// TIA Portal project "Su Tankının Doldurulup Boşaltılması_V15.1" (V15.1)
// Vorlageprojekt für das Buch mit Zielsystem S7-1200

(* hardware
DEVICE "S7-1200-Station_1"  S7-1200 Station
   slot 0: "Baugruppenträger_0"  Rack  V1.0
   slot 1: "PLC_1"  CPU 1212C DC/DC/DC  6ES7 212-1AE40-0XB0  V4.2
   slot 2: "AI 4x13BIT/AQ 2x14BIT_1"  6ES7 234-4HE32-0XB0  V2.0
DEVICE "PC-System_1"  SIMATIC PC station
   slot 0: "SIMATIC PC station"  Rail  SIMATIC PC-Station  V1.0
      slot 125: "Stationmanager"  Station_Manager  V6.0.4
   slot 1: "HMI_RT_1"  WinCC RT Advanced  6AV2 104-0xxxx-xxxx  15.1.0.0
      slot 33792: "Host interface"  Host interface
   slot 2: "IE general_1"  IE General  IE_CP  V8.2.0
*)

// ===== PLC "PLC_1"  CPU 1212C DC/DC/DC =====

VAR_GLOBAL   // PLC tag table "PLC_TAGS"
   "stop_button" AT %I0.0 : Bool;
   "start_button" AT %I0.1 : Bool;
   "sistem_devrede" AT %M5.0 : Bool;
   "set_reset_mem" AT %M5.1 : Bool;
   "sıvı_seviyesi_sensor" AT %IW30 : Int;
   "sıvı_basıncı_sensor" AT %IW32 : Int;
   "sıvı_ekle_butonu" AT %I0.3 : Bool;
   "sıvı_bosalt_butonu" AT %I0.4 : Bool;
   "Tag_1" AT %M7.1 : Bool;
   "Tag_2" AT %M7.5 : Bool;
   "Tag_3" AT %M9.0 : Bool;
END_VAR

VAR_GLOBAL   // PLC tag table "HMI_TAGS"
   "HMI_stop" AT %M6.0 : Bool;
   "HMI_start" AT %M6.1 : Bool;
   "hmi_vana_ekle" AT %QW30 : Int;
   "hmi_boşalt_boşalt" AT %QW32 : Int;
   "hmi_sıvı_ekle_butonu" AT %M7.0 : Bool;
   "hmi_sıvı_bosalt_butonu" AT %M8.2 : Bool;
END_VAR

VAR_GLOBAL   // PLC tag table "sanal_hafıza"
   "normallestırılmıs_sıvı_seviyesi_mem" AT %MD10 : Real;
   "normallestırılmıs_sıvı_basıncı_mem" AT %MD14 : Real;
   "sıvı_seviyesi" AT %MW18 : Int;
   "basınc_seviyesi" AT %MD22 : Real;
   "eklencek_sıvı_hacmi" AT %MW26 : Int;
   "boşaltılcak_sıvı_hacmi" AT %MW28 : Int;
   "kontrol_1" AT %MW8 : Int;
   "poz_mem_1" AT %M20.0 : Bool;
   "poz_mem_2" AT %M3.1 : Bool;
   "kontrol_2" AT %MW4 : Int;
END_VAR

FUNCTION "MHJ-PLC-Lab-Function-S71200" : Void   // FC9000, SCL
{ S7_Optimized_Access := 'TRUE' }
VERSION : 0.1
   VAR_TEMP
      rdTimeReturn : Int;
      outputTime : DTL;
      SyncVal : Byte;
      forVal : Int;
      forVal_2 : Int;
      Value : Byte;
   END_VAR
   VAR CONSTANT
      CompVal : Byte := 16#34;
      Value_01 : Byte := 16#11;
      Value_01_DW : DWord := 16#A165_D992;
      Value_02_DW : DWord := 16#58BE_4401;
   END_VAR
BEGIN

   #Value:=PEEK(area := 16#82,
        dbNumber := 0,
        byteOffset := 511);
   #Value := #Value + 1;

   POKE(area := 16#82,
        dbNumber := 0,
        byteOffset := 511,
        value := #Value);

   POKE(area:=16#81,
        dbNumber:=0,
        byteOffset:=1016,
        value:=#Value_01_DW);
   POKE(area := 16#81,
        dbNumber := 0,
        byteOffset := 1020,
        value := #Value_02_DW);

   POKE(area := 16#81,
        dbNumber := 0,
        byteOffset := 511,
        value := B#16#00);

   FOR #forVal := 0 TO 120 DO
       FOR #forVal_2:=0 TO 10 DO
           #rdTimeReturn:=RD_SYS_T(#outputTime);
           #rdTimeReturn := WR_SYS_T(#outputTime);
           #rdTimeReturn := RD_SYS_T(#outputTime);
           #rdTimeReturn := WR_SYS_T(#outputTime);
       END_FOR;
       #SyncVal:= PEEK(area := 16#81,
                      dbNumber := 0,
                      byteOffset := 511);
       IF #SyncVal = #CompVal THEN
          GOTO M_1;
       END_IF;
   END_FOR;
   RETURN;

   M_1:
   POKE(area := 16#81,
        dbNumber := 0,
        byteOffset := 511,
        value := B#16#0);
END_FUNCTION

ORGANIZATION_BLOCK "Main"   // OB1, LAD, ProgramCycle
TITLE = "Main Program Sweep (Cycle)"
{ S7_Optimized_Access := 'TRUE' }
VERSION : 0.1
   VAR_INPUT
      Initial_Call : Bool;   // Initial call of this OB
      Remanence : Bool;   // =True, if remanent data are available
   END_VAR
   VAR_TEMP   // added for the SCL form of the ladder/FBD networks
      _w1 : Bool;
      _w2 : Bool;
   END_VAR
BEGIN

REGION Network 1: Konnektierungsbaustein für PLC-Lab
   // Im Netzwerk 1 wird der Konnektierungsbaustein für PLC-Lab aufgerufen.
   // Dieser Aufruf darf nicht entfernt werden!
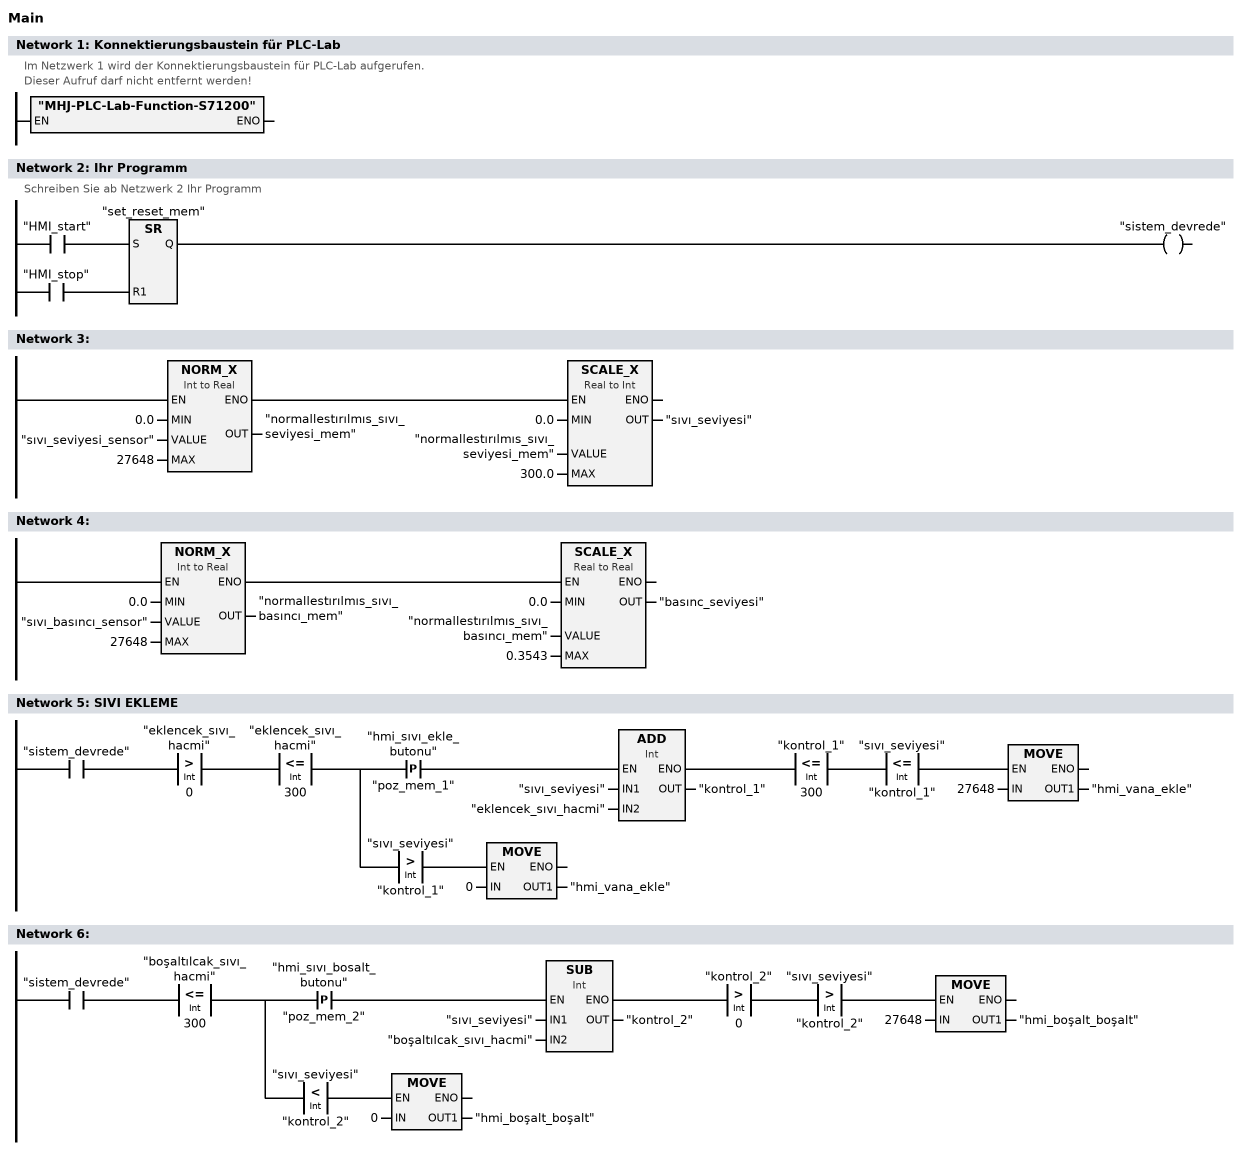
   RUNG wire#powerrail
      "MHJ-PLC-Lab-Function-S71200"()
   END_RUNG
   // the same network as SCL:
   "MHJ-PLC-Lab-Function-S71200"();
END_REGION

REGION Network 2: Ihr Programm
   // Schreiben Sie ab Netzwerk 2 Ihr Programm
   RUNG wire#powerrail
      Contact( "HMI_start" )
      S_SR(operand := "set_reset_mem", r1 := wire#w1)
      Coil( "sistem_devrede" )
   END_RUNG
   RUNG wire#powerrail
      Contact( "HMI_stop" )
   END_RUNG wire#w1
   // the same network as SCL:
   IF "HMI_start" THEN
       "set_reset_mem" := TRUE;   // SR flip-flop
   END_IF;
   IF "HMI_stop" THEN "set_reset_mem" := FALSE; END_IF;
   "sistem_devrede" := "set_reset_mem";
END_REGION

REGION Network 3
   RUNG wire#powerrail
      { S7_Templates := "[SrcType := Int, DestType := Real]" } Normalize(min := 0.0, value := "sıvı_seviyesi_sensor", max := 27648, out => "normallestırılmıs_sıvı_seviyesi_mem")
      { S7_Templates := "[SrcType := Real, DestType := Int]" } Scale(min := 0.0, value := "normallestırılmıs_sıvı_seviyesi_mem", max := 300.0, out => "sıvı_seviyesi")
   END_RUNG
   // the same network as SCL:
   "normallestırılmıs_sıvı_seviyesi_mem" := NORM_X(MIN := 0.0, VALUE := "sıvı_seviyesi_sensor", MAX := 27648);
   "sıvı_seviyesi" := SCALE_X(MIN := 0.0, VALUE := "normallestırılmıs_sıvı_seviyesi_mem", MAX := 300.0);
END_REGION

REGION Network 4
   RUNG wire#powerrail
      { S7_Templates := "[SrcType := Int, DestType := Real]" } Normalize(min := 0.0, value := "sıvı_basıncı_sensor", max := 27648, out => "normallestırılmıs_sıvı_basıncı_mem")
      { S7_Templates := "[SrcType := Real, DestType := Real]" } Scale(min := 0.0, value := "normallestırılmıs_sıvı_basıncı_mem", max := 0.3543, out => "basınc_seviyesi")
   END_RUNG
   // the same network as SCL:
   "normallestırılmıs_sıvı_basıncı_mem" := NORM_X(MIN := 0.0, VALUE := "sıvı_basıncı_sensor", MAX := 27648);
   "basınc_seviyesi" := SCALE_X(MIN := 0.0, VALUE := "normallestırılmıs_sıvı_basıncı_mem", MAX := 0.3543);
END_REGION

REGION Network 5: SIVI EKLEME
   RUNG wire#powerrail
      Contact( "sistem_devrede" )
      { S7_Templates := "SrcType := Int" } GT_Contact(in1 := "eklencek_sıvı_hacmi", in2 := 0)
      { S7_Templates := "SrcType := Int" } LE_Contact(in1 := "eklencek_sıvı_hacmi", in2 := 300)
      wire#w1
      P_Contact(operand := "hmi_sıvı_ekle_butonu", bit := "poz_mem_1")
      { S7_Templates := "SrcType := Int" } Add(in1 := "sıvı_seviyesi", in2 := "eklencek_sıvı_hacmi", out => "kontrol_1")
      { S7_Templates := "SrcType := Int" } LE_Contact(in1 := "kontrol_1", in2 := 300)
      { S7_Templates := "SrcType := Int" } LE_Contact(in1 := "sıvı_seviyesi", in2 := "kontrol_1")
      Move(in := 27648, out1 => "hmi_vana_ekle")
   END_RUNG
   RUNG wire#w1
      { S7_Templates := "SrcType := Int" } GT_Contact(in1 := "sıvı_seviyesi", in2 := "kontrol_1")
      Move(in := 0, out1 => "hmi_vana_ekle")
   END_RUNG
   // the same network as SCL:
   #_w1 := "sistem_devrede" AND ("eklencek_sıvı_hacmi" > 0) AND ("eklencek_sıvı_hacmi" <= 300);
   #_w2 := #_w1 AND "hmi_sıvı_ekle_butonu" AND NOT "poz_mem_1";   // rising edge of "hmi_sıvı_ekle_butonu"
   "poz_mem_1" := "hmi_sıvı_ekle_butonu";
   IF #_w2 THEN "kontrol_1" := "sıvı_seviyesi" + "eklencek_sıvı_hacmi"; END_IF;
   IF #_w2 AND ("kontrol_1" <= 300) AND ("sıvı_seviyesi" <= "kontrol_1") THEN
       "hmi_vana_ekle" := 27648;
   END_IF;
   IF #_w1 AND ("sıvı_seviyesi" > "kontrol_1") THEN "hmi_vana_ekle" := 0; END_IF;
END_REGION

REGION Network 6
   RUNG wire#powerrail
      Contact( "sistem_devrede" )
      { S7_Templates := "SrcType := Int" } LE_Contact(in1 := "boşaltılcak_sıvı_hacmi", in2 := 300)
      wire#w1
      P_Contact(operand := "hmi_sıvı_bosalt_butonu", bit := "poz_mem_2")
      { S7_Templates := "SrcType := Int" } Sub(in1 := "sıvı_seviyesi", in2 := "boşaltılcak_sıvı_hacmi", out => "kontrol_2")
      { S7_Templates := "SrcType := Int" } GT_Contact(in1 := "kontrol_2", in2 := 0)
      { S7_Templates := "SrcType := Int" } GT_Contact(in1 := "sıvı_seviyesi", in2 := "kontrol_2")
      Move(in := 27648, out1 => "hmi_boşalt_boşalt")
   END_RUNG
   RUNG wire#w1
      { S7_Templates := "SrcType := Int" } LT_Contact(in1 := "sıvı_seviyesi", in2 := "kontrol_2")
      Move(in := 0, out1 => "hmi_boşalt_boşalt")
   END_RUNG
   // the same network as SCL:
   #_w1 := "sistem_devrede" AND ("boşaltılcak_sıvı_hacmi" <= 300);
   #_w2 := #_w1 AND "hmi_sıvı_bosalt_butonu" AND NOT "poz_mem_2";   // rising edge of "hmi_sıvı_bosalt_butonu"
   "poz_mem_2" := "hmi_sıvı_bosalt_butonu";
   IF #_w2 THEN "kontrol_2" := "sıvı_seviyesi" - "boşaltılcak_sıvı_hacmi"; END_IF;
   IF #_w2 AND ("kontrol_2" > 0) AND ("sıvı_seviyesi" > "kontrol_2") THEN
       "hmi_boşalt_boşalt" := 27648;
   END_IF;
   IF #_w1 AND ("sıvı_seviyesi" < "kontrol_2") THEN "hmi_boşalt_boşalt" := 0; END_IF;
END_REGION
END_ORGANIZATION_BLOCK

(* ===== HMI "HMI_RT_1" =====
system functions are stored by id; their names below are inferred from use
connection "HMI_Connection_1": ETHERNET, S7_1200_OMS

HMI tags "Default tag table"
   "sıvı_seviyesi" : Int = PLC sıvı_seviyesi AT %MW18, 100 ms
   "hmi_sıvı_ekle" : Int = PLC hmi_vana_ekle AT %QW30, 100 ms
   "hmi_sıvı_boşalt" : Int = PLC hmi_boşalt_boşalt AT %QW32, 100 ms
   "sistem_devrede" : Bool = PLC sistem_devrede AT %M5.0, 100 ms
   "start_button" : Bool = PLC start_button AT %I0.1, 100 ms
   "HMI_start" : Bool = PLC HMI_start AT %M6.1, 100 ms
   "HMI_stop" : Bool = PLC HMI_stop AT %M6.0, 100 ms
   "eklencek_sıvı_hacmi" : Int = PLC eklencek_sıvı_hacmi AT %MW26, 100 ms
   "boşaltılcak_sıvı_hacmi" : Int = PLC boşaltılcak_sıvı_hacmi AT %MW28, 100 ms
   "hmi_sıvı_ekle_butonu" : Bool = PLC hmi_sıvı_ekle_butonu AT %M7.0, 100 ms
   "hmi_sıvı_bosalt_butonu" : Bool = PLC hmi_sıvı_bosalt_butonu AT %M8.2, 100 ms
   "basınc_seviyesi" : Real = PLC basınc_seviyesi AT %MD22, 100 ms

screen "Screen_1" 1024x768
   TextField "Text field_1" at 408,8 size 239x62; Text 'SU TANKI'
   GraphicView "Graphic view_1" at 152,384 size 328x319; Picture "Graphic_1"
   Bar "Bar_1" at 40,448 size 120x246; MinimumValue 0; MaximumValue 300
      ProcessValue <- "sıvı_seviyesi"
   TextField "Text field_2" at 32,96 size 207x22; Text 'SİSTEMİ BAŞLAT/DURDUR'
   Button "Button_1" at 48,144 size 64x24; TextOff 'START'
      on Press: SetBit("HMI_start")
      on Release: ResetBit("HMI_start")
   Button "Button_2" at 152,144 size 64x24; TextOff 'STOP'
      on Release: ResetBit("HMI_stop")
      on Press: SetBit("HMI_stop")
   TextField "Text field_3" at 472,464 size 81x22; Text 'SU HACMİ'
   TextField "Text field_4" at 472,520 size 144x22; Text 'SU ÇIKIŞ BASINCI'
   Circle "Circle_1" at 88,200 size 96x96
      Appearance <- "sistem_devrede"
   TextField "Text field_5" at 64,304 size 137x22; Text 'SİSTEM DEVREDE'
      Visibility <- "sistem_devrede"
   TextField "Text field_6" at 783,144 size 163x22; Text 'EKLENCEK SU HACMİ'
   TextField "Text field_7" at 784,208 size 191x22; Text 'BOŞALTILCAK SU HACMİ'
   IOField "I/O field_3" at 817,168 size 96x32; FormatPattern 999
      ProcessValue <- "eklencek_sıvı_hacmi"
   IOField "I/O field_4" at 816,232 size 96x32; FormatPattern 999
      ProcessValue <- "boşaltılcak_sıvı_hacmi"
   Button "Button_3" at 680,168 size 96x32; TextOff 'EKLE'
      on Press: SetBit("hmi_sıvı_ekle_butonu")
      on Release: ResetBit("hmi_sıvı_ekle_butonu")
   IOField "I/O field_1" at 480,488 size 96x32; FormatPattern 999
      ProcessValue <- "sıvı_seviyesi"
   IOField "I/O field_2" at 480,552 size 96x32; FormatPattern 9.999
      ProcessValue <- "basınc_seviyesi"
   Button "Button_4" at 680,232 size 96x32; TextOff 'BOSALT'
      on Press: SetBit("hmi_sıvı_bosalt_butonu")
      on Release: ResetBit("hmi_sıvı_bosalt_butonu")
*)